TYPE ModbusParOut :
STRUCT
	///寄存器字节输出
	aRcvBuffer: ARRAY[1..255] OF BYTE;
	///线圈输出		
	aRcvCoilBuffer: ARRAY[1..2000] OF BOOL;
END_STRUCT
END_TYPE

(* stored: Version 1.1.0.1, ProductVersion 3.1.4024.9
   DUT ModbusParOut: Id {021accfb-9928-4090-800e-427839aaec6a} *)
